FUNCTION TIMESTAMP_NS (* creates default a Unix-Epoch-Timestamp in nanoseconds use other start dates for other timestamp types *)
  (* Standard: 61499-1; Description: Copyright (c) 2024 Monika Wenger This program and the accompanying materials are made available under the terms of the Eclipse Public License 2.0 which is available at https://www.eclipse.org/legal/epl-2.0/ SPDX-License-Identifier: EPL-2.0 *)
  (* Version 1.0, 2024-10-14, Monika Wenger *)
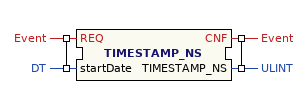
  EVENT_INPUT
    REQ WITH startDate; (* request to create a timestamp *)
  END_EVENT
  EVENT_OUTPUT
    CNF WITH TIMESTAMP_NS; (* confirms the creation of a timestamp *)
  END_EVENT
  VAR_INPUT
    startDate : DT := DT#1970-01-01-00:00:00; (* the start date used to calculate different timestamp types *)
  END_VAR
  VAR_OUTPUT
    TIMESTAMP_NS : ULINT; (* the new timestamp in nanoseconds, default Unix-Epoch *)
  END_VAR
  BODY IN ST:
FUNCTION TIMESTAMP_NS : ULINT
VAR_INPUT
	startDate : DT := DT#1970-01-01-00:00:00;
END_VAR
TIMESTAMP_NS := TIME_IN_NS_TO_ULINT(NOW() - startDate);
END_FUNCTION
  END_BODY
END_FUNCTION
